Fanuc KAREL source: NC0026.KL

-- PROVISIONAL review KL for V1013-1; original PC SHA256 ed74340a12b52c8fe95acf4d6f2a8417326735e328bb4ae22285a508c7d22332
-- Incomplete behavior may be omitted. Consult companion uncertainty JSON. Do not deploy.
PROGRAM NC0026
%NOLOCKGROUP
-- UNRESOLVED_LOCAL_POOL 1 cells at code offset 3; source declarations unknown
-- DIRECT_LOCAL_WORD_ACCESS alone does not prove INTEGER, REAL, or BOOLEAN
BEGIN
  -- UNRESOLVED_PC offsets 0-8; opcodes 2B,2C,7B
  -- UNRESOLVED_PC offsets 13-20; opcodes 9D,23
  -- UNRESOLVED_PC offsets 25-42; opcodes 21,40,41,42
  -- UNRESOLVED_PC offsets 47-64; opcodes 21,40,41,42
  -- UNRESOLVED_PC offsets 69-86; opcodes 21,40,41,42
  -- UNRESOLVED_PC offsets 91-108; opcodes 21,40,41,42
  -- UNRESOLVED_PC offsets 113-130; opcodes 21,40,41,42
  -- UNRESOLVED_PC offsets 135-152; opcodes 21,40,41,42
  -- UNRESOLVED_PC offsets 157-174; opcodes 21,40,41,42
  -- UNRESOLVED_PC offsets 179-196; opcodes 21,40,41,42
  -- UNRESOLVED_PC offsets 201-231; opcodes 21,9D,52,23,7A,40,41,42
  -- UNRESOLVED_PC offsets 236-260; opcodes 21,2E,52,23,7A,43
  -- UNRESOLVED_PC offsets 265-283; opcodes 21,2E,52,23
  -- UNRESOLVED_PC offsets 288-304; opcodes 7A,40,41,42
  -- UNRESOLVED_PC offsets 309-333; opcodes 21,2E,52,23,7A,43
  -- UNRESOLVED_PC offsets 338-356; opcodes 21,2E,52,23
  -- UNRESOLVED_PC offsets 361-377; opcodes 7A,40,41,42
  -- UNRESOLVED_PC offsets 382-406; opcodes 21,2E,52,23,7A,43
  -- UNRESOLVED_PC offsets 411-429; opcodes 21,2E,52,23
  -- UNRESOLVED_PC offsets 434-450; opcodes 7A,40,41,42
  -- UNRESOLVED_PC offsets 455-479; opcodes 21,2E,52,23,7A,43
  -- UNRESOLVED_PC offsets 484-502; opcodes 21,2E,52,23
  -- UNRESOLVED_PC offsets 507-523; opcodes 7A,40,41,42
  -- UNRESOLVED_PC offsets 528-552; opcodes 21,2E,52,23,7A,43
  -- UNRESOLVED_PC offsets 557-575; opcodes 21,2E,52,23
  -- UNRESOLVED_PC offsets 580-596; opcodes 7A,40,41,42
  -- UNRESOLVED_PC offsets 601-625; opcodes 21,2E,52,23,7A,43
  -- UNRESOLVED_PC offsets 630-648; opcodes 21,2E,52,23
  -- UNRESOLVED_PC offsets 653-669; opcodes 7A,40,41,42
  -- UNRESOLVED_PC offsets 674-698; opcodes 21,2E,52,23,7A,43
  -- UNRESOLVED_PC offsets 703-721; opcodes 21,2E,52,23
  -- UNRESOLVED_PC offsets 726-742; opcodes 7A,40,41,42
  -- UNRESOLVED_PC offsets 747-771; opcodes 21,2E,52,23,7A,43
  -- UNRESOLVED_PC offsets 776-794; opcodes 21,2E,52,23
  -- UNRESOLVED_PC offsets 804-808; opcodes 7F
  -- UNRESOLVED_PC offsets 813-817; opcodes 27,AA
  -- UNRESOLVED_PC offsets 822-826; opcodes 7F
END NC0026
